# EPICS substitutions: l2MpsLNApp/Db/mpsGC.substitutions
file "StreamGainControl.db"
{ pattern
        { DEVICE,   ATTR ,    PORT,  PARAM                           }
        { $(GC)  ,$(GCA)  , $(PORT),  DSG$(BAY)_VoltOut_$(CH)        }

}
